// TwinCAT 3 PLC project _6
// ProgramVersion: 3.1.4024.0
// libraries:
//   Tc2_MC2, * (Beckhoff Automation GmbH)
//   Tc2_NC, * (Beckhoff Automation GmbH)
//   Tc2_NcFifoAxes, * (Beckhoff Automation GmbH)
//   Tc2_Standard, * (Beckhoff Automation GmbH)
//   Tc2_System, * (Beckhoff Automation GmbH)
//   Tc2_XmlDataSrv, * (Beckhoff Automation GmbH)
//   Tc3_MC2_AdvancedHoming, * (Beckhoff Automation GmbH)
//   Tc3_Module, * (Beckhoff Automation GmbH)
//   VisuDialogs, * (System)
// project tree:
//   / GlobalTextList.TcGTLO, PlcTask.TcTTO, 视图管理器.TcVMO (not stored)
//   POUs/ MAIN.TcPOU
//   VISUs/ Visualization.TcVIS

CONFIGURATION _6
    RESOURCE PLC ON TwinCAT3
        TASK PlcTask(INTERVAL := T#10ms, PRIORITY := 21);
        PROGRAM MAIN WITH PlcTask : MAIN;
    END_RESOURCE
END_CONFIGURATION

// ---- POUs/MAIN.TcPOU
PROGRAM MAIN
VAR
	//NC PTP轴
    ACS_M1: AXIS_REF;
	ACS_M2: AXIS_REF;
	ACS_M3: AXIS_REF;
	ACS_M4: AXIS_REF;
	ACS_M5: AXIS_REF;
	ACS_M6: AXIS_REF;
	
	//FB_Enable_Axis功能块
	Enable_Axes1,Enable_Axes2,Enable_Axes3,Enable_Axes4,Enable_Axes5,Enable_Axes6: mc_power;
	ReadPosition:MC_ReadActualPosition;
	Pos1,Pos2,Pos3,Pos4,Pos5,Pos6:LREAL;
	
	is_SetPos:BOOL;
	
	//Pos[10]:LREAL;
	//Pos:ARRAY[1..6] OF LREAL;
	
	MC_JOG_ACS_M1: MC_Jog;
	MC_JOG_ACS_M2: MC_Jog;
	MC_JOG_ACS_M3: MC_Jog;
	MC_JOG_ACS_M4: MC_Jog;
	MC_JOG_ACS_M5: MC_Jog;
	MC_JOG_ACS_M6: MC_Jog;
	
	MC_SetPos_ACS_M1,MC_SetPos_ACS_M2,MC_SetPos_ACS_M3,MC_SetPos_ACS_M4,MC_SetPos_ACS_M5,MC_SetPos_ACS_M6:MC_MoveAbsolute;

	SetPos:ARRAY[1..6] OF LREAL;
	SetPosVel:LREAL ;
	Vel:ARRAY[1..6] OF LREAL;
	EnableAxes: BOOL := FALSE;
	AllAxesReady: BOOL;
	
	//JOG运动相关
	//fb_JOG_Axes: FB_JOG_Axes;
	
	JogForward_ACS_M1,JogBackward_ACS_M1: BOOL := FALSE;
	JogForward_ACS_M2,JogBackward_ACS_M2: BOOL := FALSE;
	JogForward_ACS_M3,JogBackward_ACS_M3: BOOL := FALSE;
	JogForward_ACS_M4,JogBackward_ACS_M4: BOOL := FALSE;
	JogForward_ACS_M5,JogBackward_ACS_M5: BOOL := FALSE;
	JogForward_ACS_M6,JogBackward_ACS_M6: BOOL := FALSE;

	t: INT;
	Pos_arr1,Pos_arr2: ARRAY [0..1000,1..6] OF LREAL;
	
	XmlSrvWrite: FB_XmlSrvWrite;
	sfilepath: T_MaxString:='D:\Test3.xml';
	sXPath: T_MaxString:='/dataentry/MAIN.Pos_arr1';
	writh_do: BOOL;
	XmlSrvRead: FB_XmlSrvRead;
	read_do: BOOL;	
	
	FiFo_GetDimension: FiFoGetDimension;
	fifo_display: STRING(255);

	FiFo_GroupIntegrate1,FiFo_GroupIntegrate2,FiFo_GroupIntegrate3,FiFo_GroupIntegrate4,FiFo_GroupIntegrate5,FiFo_GroupIntegrate6: FiFoGroupIntegrate;
	FiFo_SetChannelOverride: FiFoSetChannelOverride;
	FiFo_Groupout1,FiFo_Groupout2,FiFo_Groupout3,FiFo_Groupout4,FiFo_Groupout5,FiFo_Groupout6,FiFo_Disintegrate,FiFo_Override_output:st_mcoutputs;
	integrate_do: BOOL;	
	FiFo_GroupDisintegrate: FiFoGroupDisintegrate;	
	
	FiFo_Start: FiFoStart;
	start_do: BOOL;
	FiFo_Stop: FiFoStop;
	stop_do: BOOL;
	fifo_startoutput,fifo_stopoutput:st_mcoutputs;
	fifo_running:INT;
	
	pos_num:UDINT;

	FiFo_Write:FiFoWrite;
	FIFO_write_do: BOOL;
	FiFo_overWrite: FiFoOverwrite;
	FIFO_overwrite_do: BOOL;
	FIFO_write_output:st_mcoutputs;	
	
END_VAR

IF (MAIN.ACS_M1.NcToPlc.SafEntries>0) THEN
	fifo_running:= 1;
END_IF

IF (MAIN.ACS_M1.NcToPlc.SafEntries<1) THEN
	fifo_running:= 0;
END_IF


Enable_Axes1(
	Axis:= ACS_M1, 
	Enable:= EnableAxes , 
	Enable_Positive:= TRUE, 
	Enable_Negative:= TRUE, 
	Override:=15 , 
	BufferMode:= , 
	Options:= , 
	Status=> , 
	Busy=> , 
	Active=> , 
	Error=> , 
	ErrorID=> );

Enable_Axes2(
	Axis:= ACS_M2, 
	Enable:= EnableAxes , 
	Enable_Positive:= TRUE, 
	Enable_Negative:= TRUE, 
	Override:=15 , 
	BufferMode:= , 
	Options:= , 
	Status=> , 
	Busy=> , 
	Active=> , 
	Error=> , 
	ErrorID=> );
	
Enable_Axes3(
	Axis:= ACS_M3, 
	Enable:= EnableAxes , 
	Enable_Positive:= TRUE, 
	Enable_Negative:= TRUE, 
	Override:=15 , 
	BufferMode:= , 
	Options:= , 
	Status=> , 
	Busy=> , 
	Active=> , 
	Error=> , 
	ErrorID=> );
	
Enable_Axes4(
	Axis:= ACS_M4, 
	Enable:= EnableAxes , 
	Enable_Positive:= TRUE, 
	Enable_Negative:= TRUE, 
	Override:=15 , 
	BufferMode:= , 
	Options:= , 
	Status=> , 
	Busy=> , 
	Active=> , 
	Error=> , 
	ErrorID=> );
	
Enable_Axes5(
	Axis:= ACS_M5, 
	Enable:= EnableAxes , 
	Enable_Positive:= TRUE, 
	Enable_Negative:= TRUE, 
	Override:=15 , 
	BufferMode:= , 
	Options:= , 
	Status=> , 
	Busy=> , 
	Active=> , 
	Error=> , 
	ErrorID=> );

Enable_Axes6(
	Axis:= ACS_M6, 
	Enable:= EnableAxes , 
	Enable_Positive:= TRUE, 
	Enable_Negative:= TRUE, 
	Override:=15 , 
	BufferMode:= , 
	Options:= , 
	Status=> , 
	Busy=> , 
	Active=> , 
	Error=> , 
	ErrorID=> );
	
	
MC_JOG_ACS_M1(
	Axis:= ACS_M1, 
	JogForward:= JogForward_ACS_M1 , 
	JogBackwards:= JogBackward_ACS_M1 , 
	Mode:= , 
	Position:= , 
	Velocity:= , 
	Acceleration:= , 
	Deceleration:= , 
	Jerk:= , 
	Done=> , 
	Busy=> , 
	Active=> , 
	CommandAborted=> , 
	Error=> , 
	ErrorID=> );
	
MC_JOG_ACS_M2(
	Axis:= ACS_M2, 
	JogForward:= JogForward_ACS_M2 , 
	JogBackwards:= JogBackward_ACS_M2 , 
	Mode:= , 
	Position:= , 
	Velocity:= , 
	Acceleration:= , 
	Deceleration:= , 
	Jerk:= , 
	Done=> , 
	Busy=> , 
	Active=> , 
	CommandAborted=> , 
	Error=> , 
	ErrorID=> );
	
MC_JOG_ACS_M3(
	Axis:= ACS_M3, 
	JogForward:= JogForward_ACS_M3 , 
	JogBackwards:= JogBackward_ACS_M3 , 
	Mode:= , 
	Position:= , 
	Velocity:= , 
	Acceleration:= , 
	Deceleration:= , 
	Jerk:= , 
	Done=> , 
	Busy=> , 
	Active=> , 
	CommandAborted=> , 
	Error=> , 
	ErrorID=> );
	
MC_JOG_ACS_M4(
	Axis:= ACS_M4, 
	JogForward:= JogForward_ACS_M4 , 
	JogBackwards:= JogBackward_ACS_M4 , 
	Mode:= , 
	Position:= , 
	Velocity:= , 
	Acceleration:= , 
	Deceleration:= , 
	Jerk:= , 
	Done=> , 
	Busy=> , 
	Active=> , 
	CommandAborted=> , 
	Error=> , 
	ErrorID=> );
	
MC_JOG_ACS_M5(
	Axis:= ACS_M5, 
	JogForward:= JogForward_ACS_M5 , 
	JogBackwards:= JogBackward_ACS_M5 , 
	Mode:= , 
	Position:= , 
	Velocity:= , 
	Acceleration:= , 
	Deceleration:= , 
	Jerk:= , 
	Done=> , 
	Busy=> , 
	Active=> , 
	CommandAborted=> , 
	Error=> , 
	ErrorID=> );
	
MC_JOG_ACS_M6(
	Axis:= ACS_M6, 
	JogForward:= JogForward_ACS_M6 , 
	JogBackwards:= JogBackward_ACS_M6 , 
	Mode:= , 
	Position:= , 
	Velocity:= , 
	Acceleration:= , 
	Deceleration:= , 
	Jerk:= , 
	Done=> , 
	Busy=> , 
	Active=> , 
	CommandAborted=> , 
	Error=> , 
	ErrorID=> );
	

	ReadPosition(
	Axis:=ACS_M1 , 
	Enable:=TRUE , 
	Valid=> , 
	Busy=> , 
	Error=> , 
	ErrorID=> , 
	Position=>Pos1);

	ReadPosition(
	Axis:=ACS_M2 , 
	Enable:=TRUE , 
	Valid=> , 
	Busy=> , 
	Error=> , 
	ErrorID=> , 
	Position=>Pos2);
	
	ReadPosition(
	Axis:=ACS_M3 , 
	Enable:=TRUE , 
	Valid=> , 
	Busy=> , 
	Error=> , 
	ErrorID=> , 
	Position=>Pos3);
	
	ReadPosition(
	Axis:=ACS_M4 , 
	Enable:=TRUE , 
	Valid=> , 
	Busy=> , 
	Error=> , 
	ErrorID=> , 
	Position=>Pos4);
	
	ReadPosition(
	Axis:=ACS_M5 , 
	Enable:=TRUE , 
	Valid=> , 
	Busy=> , 
	Error=> , 
	ErrorID=> , 
	Position=>Pos5);
	
	ReadPosition(
	Axis:=ACS_M6 , 
	Enable:=TRUE , 
	Valid=> , 
	Busy=> , 
	Error=> , 
	ErrorID=> , 
	Position=>Pos6);
	
	
	MC_SetPos_ACS_M1(
	Axis:= ACS_M1, 
	Execute:= is_SetPos, 
	Position:= SetPos[1], 
	Velocity:=SetPosVel , 
	Acceleration:= , 
	Deceleration:= , 
	Jerk:= , 
	BufferMode:= , 
	Options:= , 
	Done=> , 
	Busy=> , 
	Active=> , 
	CommandAborted=> , 
	Error=> , 
	ErrorID=> );
	
	MC_SetPos_ACS_M2(
	Axis:= ACS_M2, 
	Execute:= is_SetPos, 
	Position:= SetPos[2], 
	Velocity:=SetPosVel , 
	Acceleration:= , 
	Deceleration:= , 
	Jerk:= , 
	BufferMode:= , 
	Options:= , 
	Done=> , 
	Busy=> , 
	Active=> , 
	CommandAborted=> , 
	Error=> , 
	ErrorID=> );
	
		MC_SetPos_ACS_M3(
	Axis:= ACS_M3, 
	Execute:= is_SetPos, 
	Position:= SetPos[3], 
	Velocity:=SetPosVel , 
	Acceleration:= , 
	Deceleration:= , 
	Jerk:= , 
	BufferMode:= , 
	Options:= , 
	Done=> , 
	Busy=> , 
	Active=> , 
	CommandAborted=> , 
	Error=> , 
	ErrorID=> );

	MC_SetPos_ACS_M4(
	Axis:= ACS_M4, 
	Execute:= is_SetPos, 
	Position:= SetPos[4], 
	Velocity:=SetPosVel , 
	Acceleration:= , 
	Deceleration:= , 
	Jerk:= , 
	BufferMode:= , 
	Options:= , 
	Done=> , 
	Busy=> , 
	Active=> , 
	CommandAborted=> , 
	Error=> , 
	ErrorID=> );

	MC_SetPos_ACS_M5(
	Axis:= ACS_M5, 
	Execute:= is_SetPos, 
	Position:= SetPos[5], 
	Velocity:=SetPosVel , 
	Acceleration:= , 
	Deceleration:= , 
	Jerk:= , 
	BufferMode:= , 
	Options:= , 
	Done=> , 
	Busy=> , 
	Active=> , 
	CommandAborted=> , 
	Error=> , 
	ErrorID=> );

	MC_SetPos_ACS_M6(
	Axis:= ACS_M6, 
	Execute:= is_SetPos, 
	Position:= SetPos[6], 
	Velocity:=SetPosVel , 
	Acceleration:= , 
	Deceleration:= , 
	Jerk:= , 
	BufferMode:= , 
	Options:= , 
	Done=> , 
	Busy=> , 
	Active=> , 
	CommandAborted=> , 
	Error=> , 
	ErrorID=> );
	
	
IF FiFo_GetDimension.iNoOfAxes=6 AND FiFo_GetDimension.iNoOfFifoEntries=50 THEN
	fifo_display:='Set Parameters Successfully,Please Continue';
ELSE
	fifo_display:='Please,Check Parameters';
END_IF

fifo();
fifo_pos();
power();
XML_write_read();


writh_do:=FALSE;
read_do:=FALSE;
FIFO_write_do:=FALSE;
FIFO_overwrite_do:=FALSE;
integrate_do:=False;

start_do:=FALSE;
stop_do:=FALSE;

FiFo_SetChannelOverride.bExecute:=FALSE;
FiFo_GroupDisintegrate.bExecute:=FALSE;

ACTION fifo:
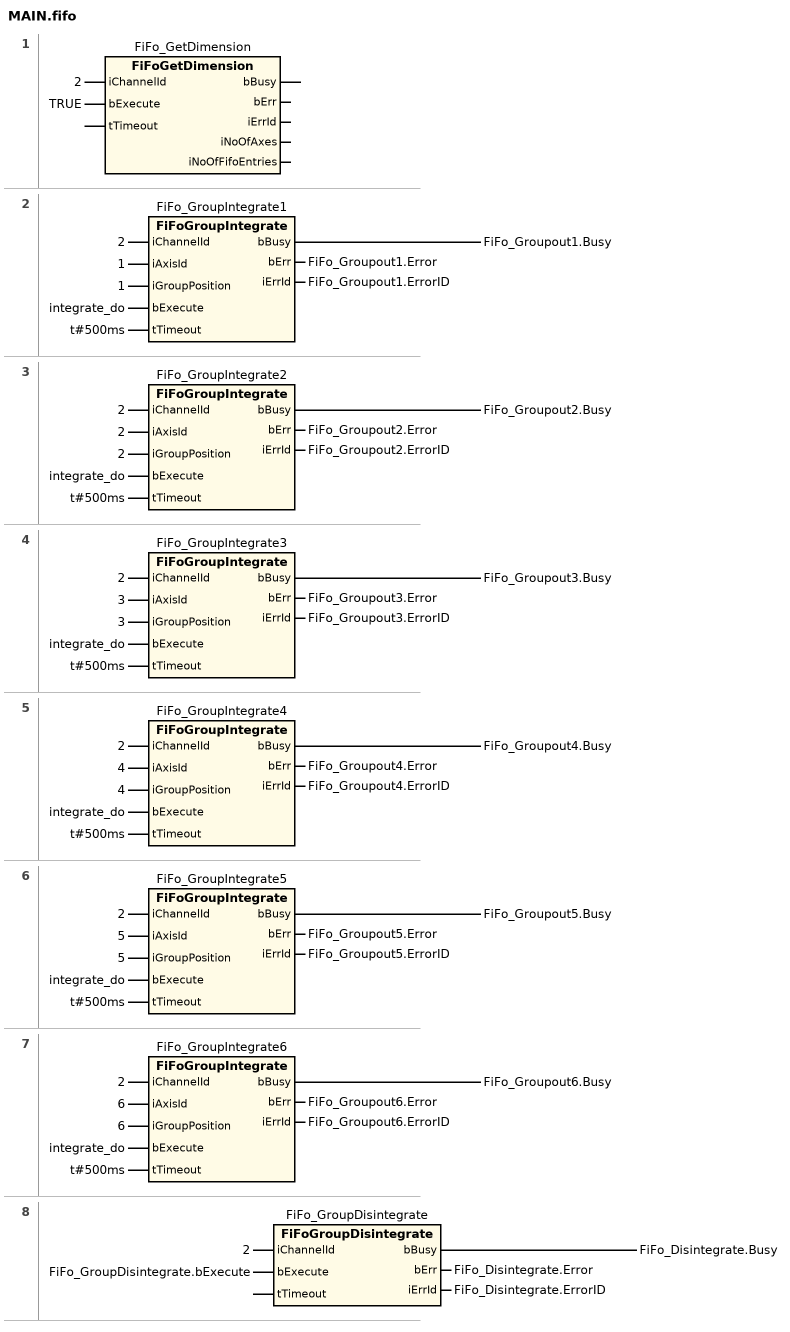
// NETWORK 1
FiFo_GetDimension(iChannelId := 2, bExecute := TRUE); // FiFoGetDimension

// NETWORK 2
FiFo_GroupIntegrate1(
    iChannelId := 2,
    iAxisId := 1,
    iGroupPosition := 1,
    bExecute := integrate_do,
    tTimeout := t#500ms,
    bErr => FiFo_Groupout1.Error,
    iErrId => FiFo_Groupout1.ErrorID); // FiFoGroupIntegrate
FiFo_Groupout1.Busy := FiFo_GroupIntegrate1.bBusy;

// NETWORK 3
FiFo_GroupIntegrate2(
    iChannelId := 2,
    iAxisId := 2,
    iGroupPosition := 2,
    bExecute := integrate_do,
    tTimeout := t#500ms,
    bErr => FiFo_Groupout2.Error,
    iErrId => FiFo_Groupout2.ErrorID); // FiFoGroupIntegrate
FiFo_Groupout2.Busy := FiFo_GroupIntegrate2.bBusy;

// NETWORK 4
FiFo_GroupIntegrate3(
    iChannelId := 2,
    iAxisId := 3,
    iGroupPosition := 3,
    bExecute := integrate_do,
    tTimeout := t#500ms,
    bErr => FiFo_Groupout3.Error,
    iErrId => FiFo_Groupout3.ErrorID); // FiFoGroupIntegrate
FiFo_Groupout3.Busy := FiFo_GroupIntegrate3.bBusy;

// NETWORK 5
FiFo_GroupIntegrate4(
    iChannelId := 2,
    iAxisId := 4,
    iGroupPosition := 4,
    bExecute := integrate_do,
    tTimeout := t#500ms,
    bErr => FiFo_Groupout4.Error,
    iErrId => FiFo_Groupout4.ErrorID); // FiFoGroupIntegrate
FiFo_Groupout4.Busy := FiFo_GroupIntegrate4.bBusy;

// NETWORK 6
FiFo_GroupIntegrate5(
    iChannelId := 2,
    iAxisId := 5,
    iGroupPosition := 5,
    bExecute := integrate_do,
    tTimeout := t#500ms,
    bErr => FiFo_Groupout5.Error,
    iErrId => FiFo_Groupout5.ErrorID); // FiFoGroupIntegrate
FiFo_Groupout5.Busy := FiFo_GroupIntegrate5.bBusy;

// NETWORK 7
FiFo_GroupIntegrate6(
    iChannelId := 2,
    iAxisId := 6,
    iGroupPosition := 6,
    bExecute := integrate_do,
    tTimeout := t#500ms,
    bErr => FiFo_Groupout6.Error,
    iErrId => FiFo_Groupout6.ErrorID); // FiFoGroupIntegrate
FiFo_Groupout6.Busy := FiFo_GroupIntegrate6.bBusy;

// NETWORK 8
FiFo_GroupDisintegrate(
    iChannelId := 2,
    bExecute := FiFo_GroupDisintegrate.bExecute,
    bErr => FiFo_Disintegrate.Error,
    iErrId => FiFo_Disintegrate.ErrorID); // FiFoGroupDisintegrate
FiFo_Disintegrate.Busy := FiFo_GroupDisintegrate.bBusy;

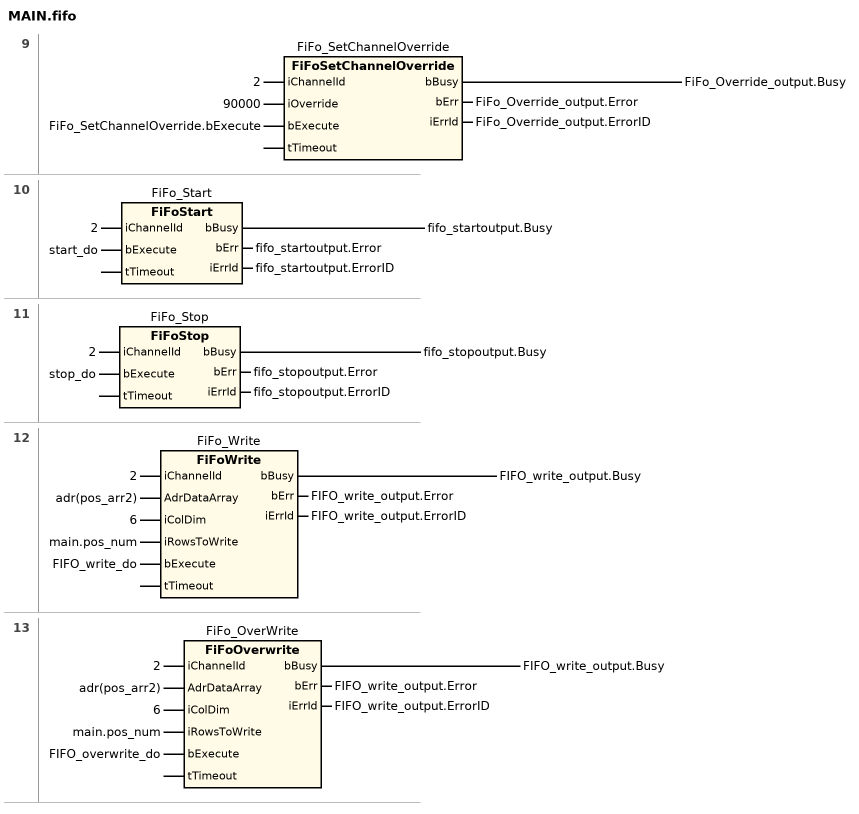
// NETWORK 9
FiFo_SetChannelOverride(
    iChannelId := 2,
    iOverride := 90000,
    bExecute := FiFo_SetChannelOverride.bExecute,
    bErr => FiFo_Override_output.Error,
    iErrId => FiFo_Override_output.ErrorID); // FiFoSetChannelOverride
FiFo_Override_output.Busy := FiFo_SetChannelOverride.bBusy;

// NETWORK 10
FiFo_Start(
    iChannelId := 2,
    bExecute := start_do,
    bErr => fifo_startoutput.Error,
    iErrId => fifo_startoutput.ErrorID); // FiFoStart
fifo_startoutput.Busy := FiFo_Start.bBusy;

// NETWORK 11
FiFo_Stop(
    iChannelId := 2,
    bExecute := stop_do,
    bErr => fifo_stopoutput.Error,
    iErrId => fifo_stopoutput.ErrorID); // FiFoStop
fifo_stopoutput.Busy := FiFo_Stop.bBusy;

// NETWORK 12
FiFo_Write(
    iChannelId := 2,
    AdrDataArray := adr(pos_arr2),
    iColDim := 6,
    iRowsToWrite := main.pos_num,
    bExecute := FIFO_write_do,
    bErr => FIFO_write_output.Error,
    iErrId => FIFO_write_output.ErrorID); // FiFoWrite
FIFO_write_output.Busy := FiFo_Write.bBusy;

// NETWORK 13
FiFo_OverWrite(
    iChannelId := 2,
    AdrDataArray := adr(pos_arr2),
    iColDim := 6,
    iRowsToWrite := main.pos_num,
    bExecute := FIFO_overwrite_do,
    bErr => FIFO_write_output.Error,
    iErrId => FIFO_write_output.ErrorID); // FiFoOverwrite
FIFO_write_output.Busy := FiFo_OverWrite.bBusy;
END_ACTION

ACTION fifo_pos:
FOR t:=0 TO 50 BY 1 DO
	Pos_arr1[t,1]:=0;
	Pos_arr1[t,2]:=0;
	Pos_arr1[t,3]:=0;
	
	Pos_arr1[t,4]:=0;
	Pos_arr1[t,5]:=0;
	Pos_arr1[t,6]:=60*SIN(0.0628*t);
END_FOR
END_ACTION

ACTION power:
ACS_M1.PlcToNc.ControlDWord:=7;
ACS_M2.PlcToNc.ControlDWord:=7;
ACS_M3.PlcToNc.ControlDWord:=7;
ACS_M4.PlcToNc.ControlDWord:=7;
ACS_M5.PlcToNc.ControlDWord:=7;
ACS_M6.PlcToNc.ControlDWord:=7;

ACS_M1.PlcToNc.Override:=1000000;
ACS_M2.PlcToNc.Override:=1000000;
ACS_M3.PlcToNc.Override:=1000000;
ACS_M4.PlcToNc.Override:=1000000;
ACS_M5.PlcToNc.Override:=1000000;
ACS_M6.PlcToNc.Override:=1000000;
END_ACTION

ACTION XML_write_read:
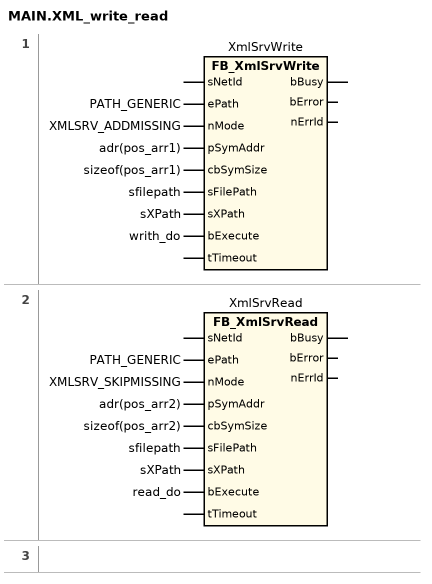
// NETWORK 1
XmlSrvWrite(
    ePath := PATH_GENERIC,
    nMode := XMLSRV_ADDMISSING,
    pSymAddr := adr(pos_arr1),
    cbSymSize := sizeof(pos_arr1),
    sFilePath := sfilepath,
    sXPath := sXPath,
    bExecute := writh_do); // FB_XmlSrvWrite

// NETWORK 2
XmlSrvRead(
    ePath := PATH_GENERIC,
    nMode := XMLSRV_SKIPMISSING,
    pSymAddr := adr(pos_arr2),
    cbSymSize := sizeof(pos_arr2),
    sFilePath := sfilepath,
    sXPath := sXPath,
    bExecute := read_do); // FB_XmlSrvRead

// NETWORK 3
END_ACTION

END_PROGRAM

// ---- GlobalTextList.TcGTLO
TEXTLIST GlobalTextList
  190 = '%.2f'
  525 = '%2f'
  291 = '%d'
  269 = '%s'
  195 = '132'
  813 = 'axis1_buffer%d'
  277 = 'BASIC'
  965 = 'disintergrate'
  594 = 'FIFO'
  823 = 'fifo_overwrtie'
  946 = 'fifo_write'
  533 = 'INTERGRATE'
  827 = 'intergrate'
  608 = 'JOG+'
  109 = 'JOG-'
  499 = 'SetChannelOverride'
  830 = 'start'
  705 = 'stop'
  755 = 'xml_read'
  777 = 'xml_write'
  104 = '位置数据量：%d'
  658 = '使能'
  137 = '失能'
  124 = '实际'
  746 = '期望速度'
  55 = '目标'
  981 = '轴一'
  366 = '轴三'
  539 = '轴二'
  155 = '轴五'
  75 = '轴六'
  733 = '轴四'
  299 = '轴数量：%.2f'
  493 = '轴数量：%d'
  544 = '运动到目标'
END_TEXTLIST

// ---- VISUs/Visualization.TcVIS
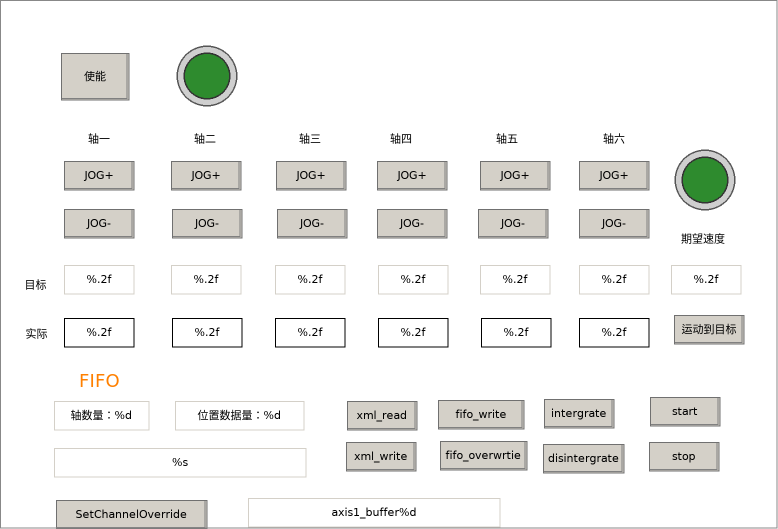
VISUALIZATION Visualization  // 778x529
    Button (61,53 68x47), "使能"
        OnMouseClick: execute { MAIN.EnableAxes := Not MAIN.EnableAxes }
    Lamp1 (172,41 70x70), variable: MAIN.Enable_Axes1.Status, style: Lamp-Lamp1-Green
    Button (64,161 70x29), "JOG+"
        OnMouseDown: execute { MAIN.JogForward_ACS_M1 := True }
        OnMouseUp: execute { MAIN.JogForward_ACS_M1 := FALSE }
    Button (171,161 70x29), "JOG+"
        OnMouseDown: execute { MAIN.JogForward_ACS_M2 := True }
        OnMouseUp: execute { MAIN.JogForward_ACS_M2 := FALSE }
    Button (276,161 70x29), "JOG+"
        OnMouseDown: execute { MAIN.JogForward_ACS_M3 := True }
        OnMouseUp: execute { MAIN.JogForward_ACS_M3 := false }
    Button (377,161 70x29), "JOG+"
        OnMouseDown: execute { MAIN.JogForward_ACS_M4 := True }
        OnMouseUp: execute { MAIN.JogForward_ACS_M4 :=false }
    Button (579,161 70x29), "JOG+"
        OnMouseDown: execute { MAIN.JogForward_ACS_M6 :=TRUE }
        OnMouseUp: execute { MAIN.JogForward_ACS_M6 :=false }
    Button (480,161 70x29), "JOG+"
        OnMouseDown: execute { MAIN.JogForward_ACS_M5 := True }
        OnMouseUp: execute { MAIN.JogForward_ACS_M5 :=false }
    Button (64,209 70x29), "JOG-"
        OnMouseDown: execute { MAIN.JogBackward_ACS_M1 := TRUE }
        OnMouseUp: execute { MAIN.JogBackward_ACS_M1:=FALSE }
    Label (24,124 150x30), "轴一"
    Label (235,124 150x30), "轴三"
    Label (130,124 150x30), "轴二"
    Label (326,124 150x30), "轴四"
    Label (432,124 150x30), "轴五"
    Label (539,124 150x30), "轴六"
    Textfield (64,265 70x29), "%.2f", text variable: MAIN.SetPos[1]
        OnMouseClick: write MAIN.SetPos[1] via Default
    Label (7,270 57x30), "目标"
    Label (8,319 57x30), "实际"
    Rectangle (64,318 70x29), "%.2f", text variable: MAIN.Pos1
    Rectangle (172,318 70x29), "%.2f", text variable: MAIN.Pos2
    Rectangle (378,318 70x29), "%.2f", text variable: MAIN.Pos4
    Rectangle (579,318 70x29), "%.2f", text variable: MAIN.Pos6
    Rectangle (275,318 70x29), "%.2f", text variable: MAIN.Pos3
    Rectangle (481,318 70x29), "%.2f", text variable: MAIN.Pos5
    Button (674,315 70x29), "运动到目标"
        OnMouseClick: execute { MAIN.is_SetPos:= NOT Main.is_SetPos }
    Button (172,209 70x29), "JOG-"
        OnMouseDown: execute { MAIN.JogBackward_ACS_M2 := TRUE }
        OnMouseUp: execute { MAIN.JogBackward_ACS_M2:=FALSE }
    Button (277,209 70x29), "JOG-"
        OnMouseDown: execute { MAIN.JogBackward_ACS_M3 := TRUE }
        OnMouseUp: execute { MAIN.JogBackward_ACS_M3:=FALSE }
    Button (377,209 70x29), "JOG-"
        OnMouseDown: execute { MAIN.JogBackward_ACS_M4 := TRUE }
        OnMouseUp: execute { MAIN.JogBackward_ACS_M4:=FALSE }
    Button (478,209 70x29), "JOG-"
        OnMouseDown: execute { MAIN.JogBackward_ACS_M5 := TRUE }
        OnMouseUp: execute { MAIN.JogBackward_ACS_M5:=FALSE }
    Button (579,209 70x29), "JOG-"
        OnMouseDown: execute { MAIN.JogBackward_ACS_M6 := TRUE }
        OnMouseUp: execute { MAIN.JogBackward_ACS_M6:=FALSE }
    Lamp1 (670,145 70x70), variable: MAIN.is_SetPos, style: Lamp-Lamp1-Green
    Textfield (579,265 70x29), "%.2f", text variable: MAIN.SetPos[6]
        OnMouseClick: write MAIN.SetPos[6] via Default
    Textfield (480,265 70x29), "%.2f", text variable: MAIN.SetPos[5]
        OnMouseClick: write MAIN.SetPos[5] via Default
    Textfield (275,265 70x29), "%.2f", text variable: MAIN.SetPos[3]
        OnMouseClick: write MAIN.SetPos[3] via Default
    Textfield (378,265 70x29), "%.2f", text variable: MAIN.SetPos[4]
        OnMouseClick: write MAIN.SetPos[4] via Default
    Textfield (171,265 70x29), "%.2f", text variable: MAIN.SetPos[2]
        OnMouseClick: write MAIN.SetPos[2] via Default
    Textfield (671,265 70x29), "%.2f", text variable: MAIN.SetPosVel
        OnMouseClick: write MAIN.SetPosVel via Default
    Label (628,224 150x30), "期望速度"
    Label (52,366 95x30), "FIFO"
    Textfield (54,401 95x29), "轴数量：%d", text variable: MAIN.FiFo_GetDimension.iNoOfAxes
    Textfield (175,401 129x29), "位置数据量：%d", text variable: MAIN.FiFo_GetDimension.iNoOfFifoEntries
    Textfield (54,448 252x29), "%s", text variable: MAIN.fifo_display
    Button (347,401 70x29), "xml_read", text variable: MAIN.read_do
        OnMouseClick: execute { MAIN.read_do:=true }
    Button (346,442 70x29), "xml_write", text variable: MAIN.writh_do
        OnMouseClick: execute { MAIN.writh_do:= true }
    Button (438,400 86x29), "fifo_write", text variable: MAIN.FIFO_write_do
        OnMouseClick: execute { main.FIFO_write_do:=true; }
    Button (440,441 87x29), "fifo_overwrtie", text variable: MAIN.FIFO_overwrite_do
        OnMouseClick: execute { main.FIFO_overwrite_do:=true; }
    Button (649,442 70x29), "stop", text variable: MAIN.stop_do
        OnMouseClick: execute { main.stop_do:=true }
    Button (650,397 70x29), "start", text variable: MAIN.start_do
        OnMouseClick: execute { main.start_do:=true }
    Button (543,444 81x29), "disintergrate", text variable: MAIN.FiFo_GroupDisintegrate
        OnMouseClick: execute { main.FiFo_GroupDisintegrate.bExecute:=true }
    Button (544,399 70x29), "intergrate", text variable: MAIN.integrate_do
        OnMouseClick: execute { main.integrate_do:=true }
    Button (56,500 151x29), "SetChannelOverride", text variable: MAIN.FiFo_SetChannelOverride
        OnMouseClick: execute { main.FiFo_SetChannelOverride.bExecute:=true }
    Textfield (248,498 252x29), "axis1_buffer%d", text variable: MAIN.ACS_M1.NcToPlc.SafEntries
END_VISUALIZATION
